(* PLC project I2C sensor modules Function Blocks, OpenPLC Arduino Function Blocks Library 1.0, author Sakunamary Xiao *)
(* stored: creationDateTime 2023-8-1T02:33:11, modificationDateTime 2023-8-1T02:33:11 *)

(* Reads temperature from I2C module *)
FUNCTION_BLOCK I2C_THREMO_4_OUT
  VAR_INPUT
    ADDR_SLAVE : INT;  (* I2C module address *)
    SCK_PIN : INT;  (* I2C module SCK PIN *)
    SDA_PIN : INT;  (* I2C module SDA PIN *)
  END_VAR
  VAR_OUTPUT
    OUT_0 : REAL;  (* Temperature output in Celsius *)
    OUT_1 : REAL;  (* Temperature output in Celsius *)
    OUT_2 : REAL;  (* Temperature output in Celsius *)
    OUT_3 : REAL;  (* Temperature output in Celsius *)
  END_VAR

            OUT := 0.0;
          
END_FUNCTION_BLOCK

(* Reads Temperature and Humidity from I2C module *)
FUNCTION_BLOCK I2C_AHT20
  VAR_INPUT
    SCK_PIN : INT;  (* I2C module SCK PIN *)
    SDA_PIN : INT;  (* I2C module SDA PIN *)
  END_VAR
  VAR_OUTPUT
    TEMP : REAL;  (* Temperature output in Celsius *)
    RH : REAL;  (* Humidity output *)
  END_VAR

            OUT := 0.0;
          
END_FUNCTION_BLOCK
